(* Logix 5000 project; controller R5_CSS vendor 1 type 14 code 74 rev 19.11; software revision 19.01; part 13 of 20 *)
(* tags used below, declared in another part *)
   AC102A : ANALYTICAL;   // QUENCH WATER CONDUCTIVITY CONTROL
   bryans_Test4 : BOOL;
   CSS_Heartbeat : BOOL;
   CSS_OK_TO_RUN : BOOL;   // PRU_RUN_DISABLE 0 = Cannot Run 1 = OK to Run
   CSS_OK_TO_START : BOOL;   // PRU_START_DISABLE 0 = Cannot Start 1 = OK to Start
   LC303A : LEVEL_CONTROL;   // AQUEOUS PHASE OF PRIMARY SETTLER
   LC304 : LEVEL_CONTROL;   // SETTLER SECONDARY TANK INTERFACE LEVEL
   P101A : PUMP_CONTROL;
   P101B : PUMP_CONTROL;
   PC408 : PRESSURE_CONTROL;
   PRU_BLOWER_SEQ : INT;   // PRU BLOWER SEQUENCE NUMBER
   PRU_DELAY_REQ : INT;
   PRU_MaxTempDelayMin : REAL;
   PRU_MaxTempDelta : REAL;
   PRU_PT404 : REAL[10];
   PRU_PT404_Done : REAL[10];
   PRU_PT404_Max : REAL[10];
   PRU_RECIPE_LOAD : INT;
   PRU_RECIPE_LOAD_DLY : TIMER[10];
   PRU_RunDoneTemp : BOOL[32];
   PRU_RunDoneTime : BOOL[32];
   PRU_Running : BOOL[32];
   PRU_RunningMaxHrs : REAL;
   PRU_RunningMaxTempDelay : TIMER[10];
   PRU_RunningMinutePulse : TIMER[10];
   PRU_RunningTotalMin : COUNTER[10];
   PRU_START_REQ : INT;
   PRU_STARTDISABLE : DINT;   // PRU START DISABLE
   PRUA_CHANGE : INT;
   PRUA_CHANGE_OF_STATE : BOOL;
   PRUA_COMMS_TIMER : TIMER;
   PRUA_ECOOL : BOOL;
   PRUA_ECOOL_TON : TIMER;
   PRUA_HeartbeatCommsLoss : BOOL;
   PRUA_HeartbeatOffONS : BOOL;
   PRUA_HeartbeatOnONS : BOOL;
   PRUA_READ : INT[30];
   PRUA_START_REQ_ONS : BOOL[32];
   PRUA_WRITE : INT[40];
   PRUB_CHANGE : INT;
   PRUB_CHANGE_OF_STATE : BOOL;
   PRUB_COMMS_TIMER : TIMER;
   PRUB_ECOOL : BOOL;
   PRUB_ECOOL_TON : TIMER;
   PRUB_HeartbeatCommsLoss : BOOL;
   PRUB_HeartbeatOffONS : BOOL;
   PRUB_HeartbeatOnONS : BOOL;
   PRUB_READ : INT[30];
   PRUB_START_REQ_ONS : BOOL[32];
   PRUB_WRITE : INT[40];
   PRUC_CHANGE : INT;
   PRUC_CHANGE_OF_STATE : BOOL;
   PRUC_COMMS_TIMER : TIMER;
   PRUC_ECOOL : BOOL;
   PRUC_ECOOL_TON : TIMER;
   PRUC_HeartbeatCommsLoss : BOOL;
   PRUC_HeartbeatOffONS : BOOL;
   PRUC_HeartbeatOnONS : BOOL;
   PRUC_READ : INT[30];
   PRUC_START_REQ_ONS : BOOL[32];
   PRUC_WRITE : INT[40];
   TC101A : TEMP_CONTROL;   // QUENCH BASIN TRANSFER BASIN A TEMPERATURE CONTROL
   TC321A : TEMP_CONTROL;   // COALESCER OIL CHAMBER TRANSFER PUMP A TEMPERATURE TRANSMITTER
   TC321B : TEMP_CONTROL;   // COALESCER OIL CHAMBER TRANSFER PUMP B TEMPERATURE TRANSMITTER
   TMR_FAULT : DINT;
   UTL_Comms : DINT[3];
   UTL_CommsLossAlm : BOOL;
(* MainProgram, continued *)

ROUTINE PC408_FILL_IN_HERE   (* ladder *)
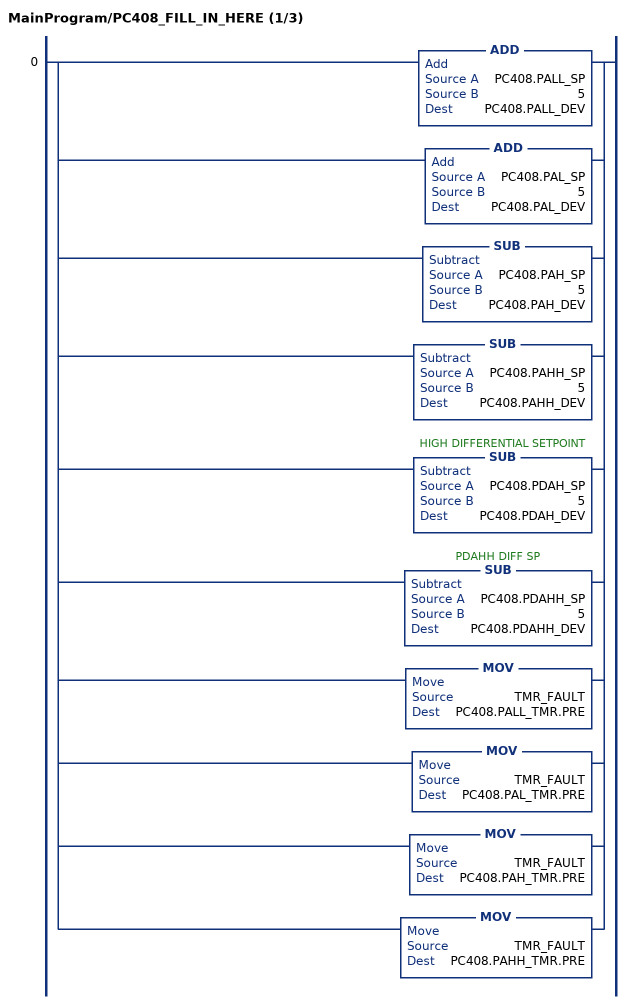
   0: [ADD(PC408.PALL_SP,5,PC408.PALL_DEV) ,ADD(PC408.PAL_SP,5,PC408.PAL_DEV) ,SUB(PC408.PAH_SP,5,PC408.PAH_DEV) ,SUB(PC408.PAHH_SP,5,PC408.PAHH_DEV) ,SUB(PC408.PDAH_SP,5,PC408.PDAH_DEV) ,SUB(PC408.PDAHH_SP,5,PC408.PDAHH_DEV) ,MOV(TMR_FAULT,PC408.PALL_TMR.PRE) ,MOV(TMR_FAULT,PC408.PAL_TMR.PRE) ,MOV(TMR_FAULT,PC408.PAH_TMR.PRE) ,MOV(TMR_FAULT,PC408.PAHH_TMR.PRE) ];
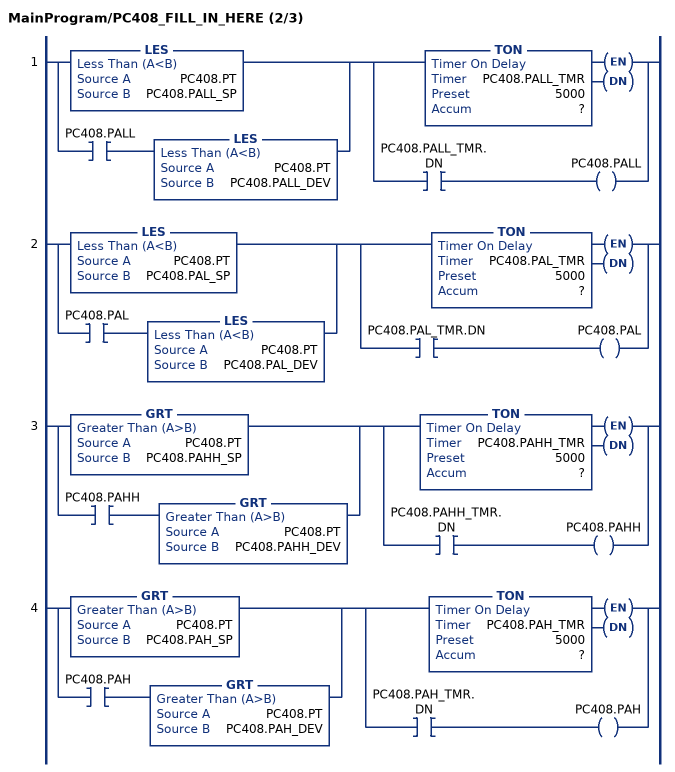
   1: [LES(PC408.PT,PC408.PALL_SP) ,XIC(PC408.PALL) LES(PC408.PT,PC408.PALL_DEV) ][TON(PC408.PALL_TMR,?,?) ,XIC(PC408.PALL_TMR.DN) OTE(PC408.PALL) ];
   2: [LES(PC408.PT,PC408.PAL_SP) ,XIC(PC408.PAL) LES(PC408.PT,PC408.PAL_DEV) ][TON(PC408.PAL_TMR,?,?) ,XIC(PC408.PAL_TMR.DN) OTE(PC408.PAL) ];
   3: [GRT(PC408.PT,PC408.PAHH_SP) ,XIC(PC408.PAHH) GRT(PC408.PT,PC408.PAHH_DEV) ][TON(PC408.PAHH_TMR,?,?) ,XIC(PC408.PAHH_TMR.DN) OTE(PC408.PAHH) ];
   4: [GRT(PC408.PT,PC408.PAH_SP) ,XIC(PC408.PAH) GRT(PC408.PT,PC408.PAH_DEV) ][TON(PC408.PAH_TMR,?,?) ,XIC(PC408.PAH_TMR.DN) OTE(PC408.PAH) ];
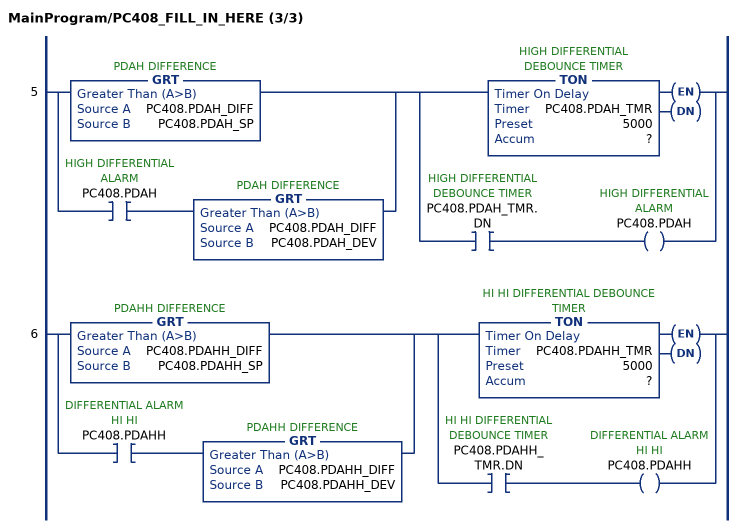
   5: [GRT(PC408.PDAH_DIFF,PC408.PDAH_SP) ,XIC(PC408.PDAH) GRT(PC408.PDAH_DIFF,PC408.PDAH_DEV) ][TON(PC408.PDAH_TMR,?,?) ,XIC(PC408.PDAH_TMR.DN) OTE(PC408.PDAH) ];
   6: [GRT(PC408.PDAHH_DIFF,PC408.PDAHH_SP) ,XIC(PC408.PDAHH) GRT(PC408.PDAHH_DIFF,PC408.PDAHH_DEV) ][TON(PC408.PDAHH_TMR,?,?) ,XIC(PC408.PDAHH_TMR.DN) OTE(PC408.PDAHH) ];
END_ROUTINE

ROUTINE PRU_STRTDIS   (* ladder *)
// PRU START DISABLE LOGIC
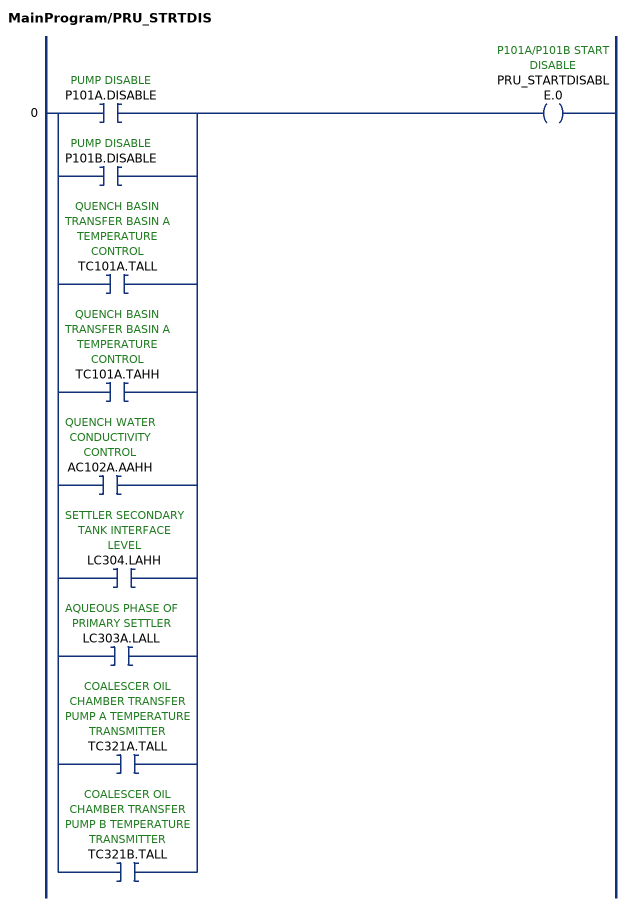
   0: [XIC(P101A.DISABLE) ,XIC(P101B.DISABLE) ,XIC(TC101A.TALL) ,XIC(TC101A.TAHH) ,XIC(AC102A.AAHH) ,XIC(LC304.LAHH) ,XIC(LC303A.LALL) ,XIC(TC321A.TALL) ,XIC(TC321B.TALL) ]OTE(PRU_STARTDISABLE.0);
END_ROUTINE

ROUTINE PRUA   (* ladder *)
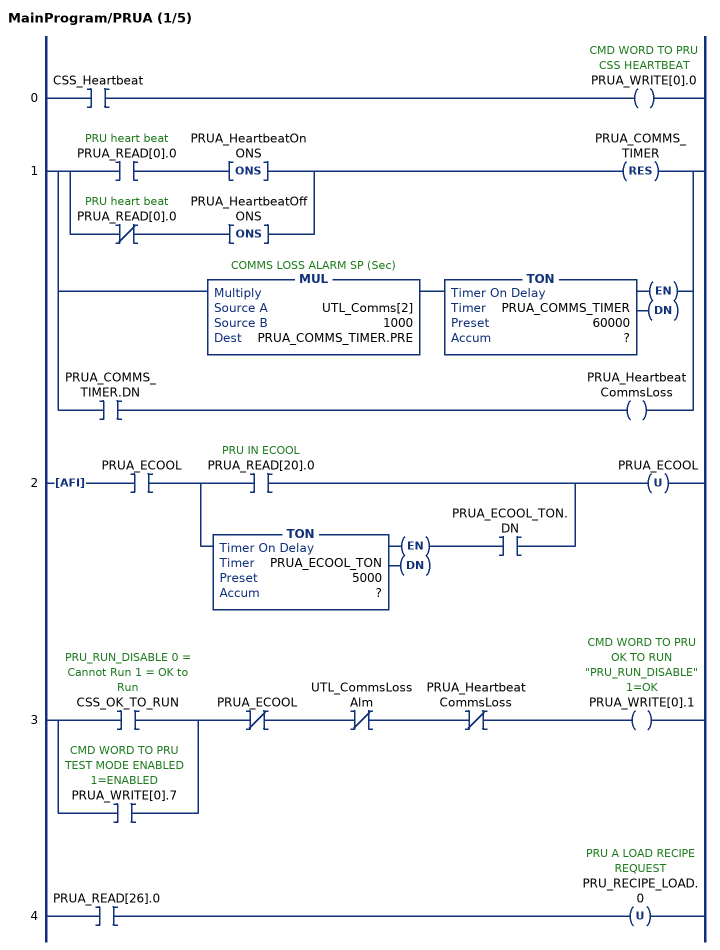
   0: XIC(CSS_Heartbeat)OTE(PRUA_WRITE[0].0);
   1: [[XIC(PRUA_READ[0].0) ONS(PRUA_HeartbeatOnONS) ,XIO(PRUA_READ[0].0) ONS(PRUA_HeartbeatOffONS) ] RES(PRUA_COMMS_TIMER) ,MUL(UTL_Comms[2],1000,PRUA_COMMS_TIMER.PRE) TON(PRUA_COMMS_TIMER,?,?) ,XIC(PRUA_COMMS_TIMER.DN) OTE(PRUA_HeartbeatCommsLoss) ];
   2: AFI()XIC(PRUA_ECOOL)[XIC(PRUA_READ[20].0) ,TON(PRUA_ECOOL_TON,?,?) XIC(PRUA_ECOOL_TON.DN) ]OTU(PRUA_ECOOL);
   3: [XIC(CSS_OK_TO_RUN) ,XIC(PRUA_WRITE[0].7) ]XIO(PRUA_ECOOL)XIO(UTL_CommsLossAlm)XIO(PRUA_HeartbeatCommsLoss)OTE(PRUA_WRITE[0].1);
   4: XIC(PRUA_READ[26].0)OTU(PRU_RECIPE_LOAD.0);
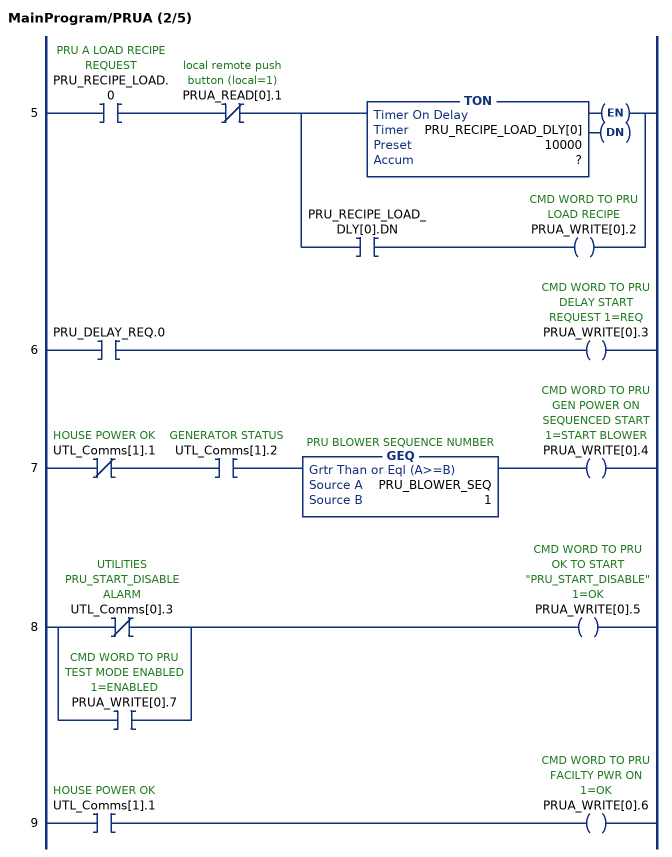
   5: XIC(PRU_RECIPE_LOAD.0)XIO(PRUA_READ[0].1)[TON(PRU_RECIPE_LOAD_DLY[0],?,?) ,XIC(PRU_RECIPE_LOAD_DLY[0].DN) OTE(PRUA_WRITE[0].2) ];
   6: XIC(PRU_DELAY_REQ.0)OTE(PRUA_WRITE[0].3);
   7: XIO(UTL_Comms[1].1)XIC(UTL_Comms[1].2)GEQ(PRU_BLOWER_SEQ,1)OTE(PRUA_WRITE[0].4);
   8: [XIO(UTL_Comms[0].3) ,XIC(PRUA_WRITE[0].7) ]OTE(PRUA_WRITE[0].5);
   9: XIC(UTL_Comms[1].1)OTE(PRUA_WRITE[0].6);
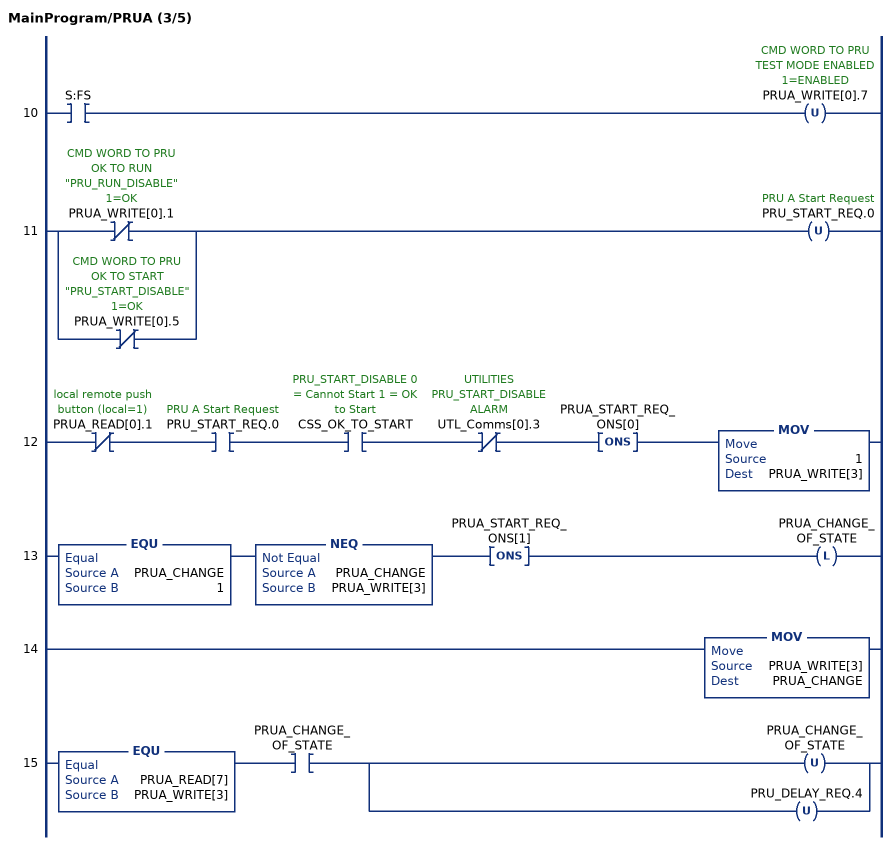
   10: XIC(S:FS)OTU(PRUA_WRITE[0].7);
   11: [XIO(PRUA_WRITE[0].1) ,XIO(PRUA_WRITE[0].5) ]OTU(PRU_START_REQ.0);
   12: XIO(PRUA_READ[0].1)XIC(PRU_START_REQ.0)XIC(CSS_OK_TO_START)XIO(UTL_Comms[0].3)ONS(PRUA_START_REQ_ONS[0])MOV(1,PRUA_WRITE[3]);
   13: EQU(PRUA_CHANGE,1)NEQ(PRUA_CHANGE,PRUA_WRITE[3])ONS(PRUA_START_REQ_ONS[1])OTL(PRUA_CHANGE_OF_STATE);
   14: MOV(PRUA_WRITE[3],PRUA_CHANGE);
   15: EQU(PRUA_READ[7],PRUA_WRITE[3])XIC(PRUA_CHANGE_OF_STATE)[OTU(PRUA_CHANGE_OF_STATE) ,OTU(PRU_DELAY_REQ.4) ];
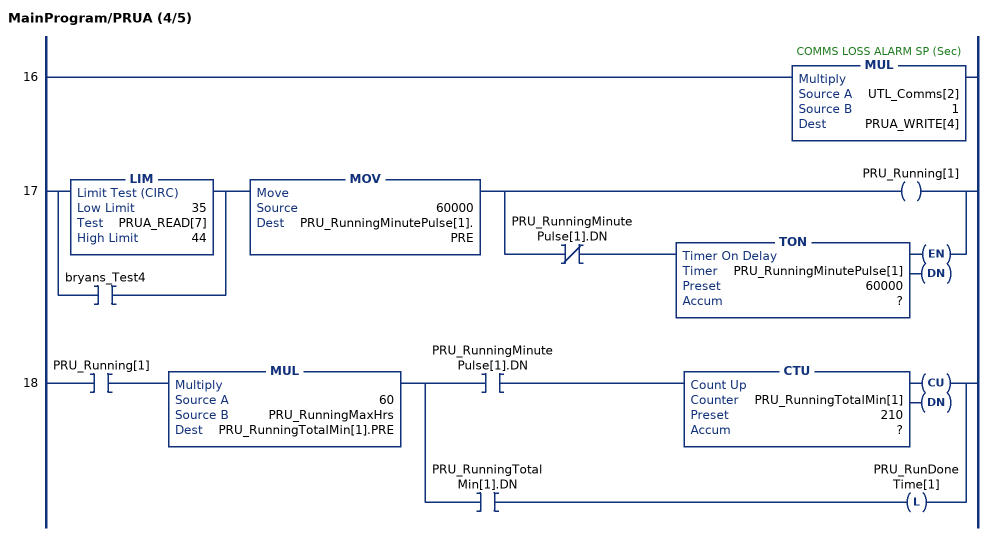
   16: MUL(UTL_Comms[2],1,PRUA_WRITE[4]);
   17: [LIM(35,PRUA_READ[7],44) ,XIC(bryans_Test4) ]MOV(60000,PRU_RunningMinutePulse[1].PRE)[OTE(PRU_Running[1]) ,XIO(PRU_RunningMinutePulse[1].DN) TON(PRU_RunningMinutePulse[1],?,?) ];
   18: XIC(PRU_Running[1])MUL(60,PRU_RunningMaxHrs,PRU_RunningTotalMin[1].PRE)[XIC(PRU_RunningMinutePulse[1].DN) CTU(PRU_RunningTotalMin[1],?,?) ,XIC(PRU_RunningTotalMin[1].DN) OTL(PRU_RunDoneTime[1]) ];
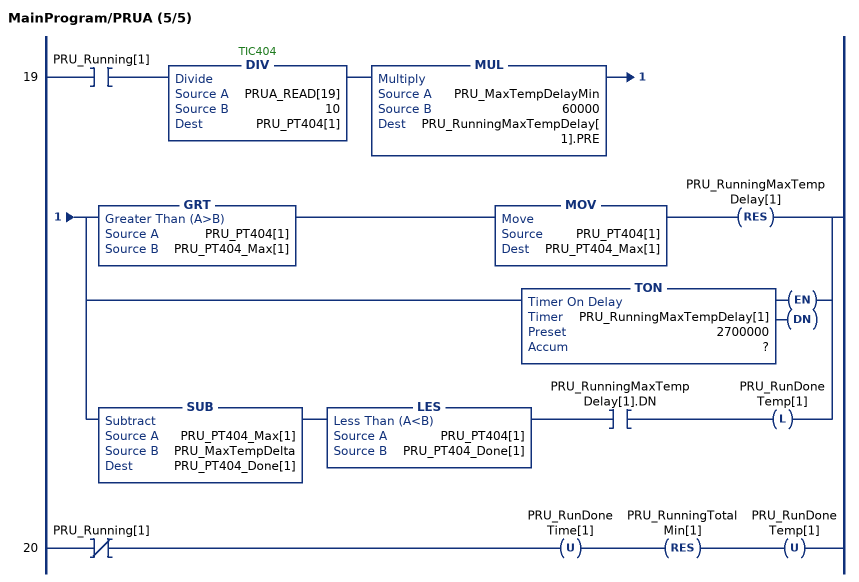
   19: XIC(PRU_Running[1])DIV(PRUA_READ[19],10,PRU_PT404[1])MUL(PRU_MaxTempDelayMin,60000,PRU_RunningMaxTempDelay[1].PRE)[GRT(PRU_PT404[1],PRU_PT404_Max[1]) MOV(PRU_PT404[1],PRU_PT404_Max[1]) RES(PRU_RunningMaxTempDelay[1]) ,TON(PRU_RunningMaxTempDelay[1],?,?) ,SUB(PRU_PT404_Max[1],PRU_MaxTempDelta,PRU_PT404_Done[1]) LES(PRU_PT404[1],PRU_PT404_Done[1]) XIC(PRU_RunningMaxTempDelay[1].DN) OTL(PRU_RunDoneTemp[1]) ];
   20: XIO(PRU_Running[1])OTU(PRU_RunDoneTime[1])RES(PRU_RunningTotalMin[1])OTU(PRU_RunDoneTemp[1]);
END_ROUTINE

ROUTINE PRUB   (* ladder *)
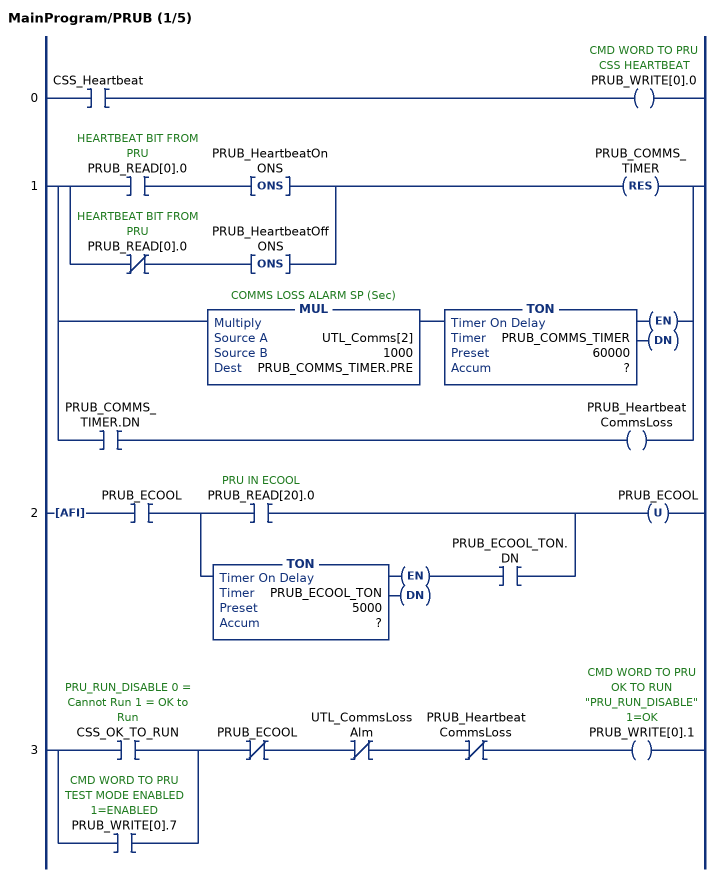
   0: XIC(CSS_Heartbeat)OTE(PRUB_WRITE[0].0);
   1: [[XIC(PRUB_READ[0].0) ONS(PRUB_HeartbeatOnONS) ,XIO(PRUB_READ[0].0) ONS(PRUB_HeartbeatOffONS) ] RES(PRUB_COMMS_TIMER) ,MUL(UTL_Comms[2],1000,PRUB_COMMS_TIMER.PRE) TON(PRUB_COMMS_TIMER,?,?) ,XIC(PRUB_COMMS_TIMER.DN) OTE(PRUB_HeartbeatCommsLoss) ];
   2: AFI()XIC(PRUB_ECOOL)[XIC(PRUB_READ[20].0) ,TON(PRUB_ECOOL_TON,?,?) XIC(PRUB_ECOOL_TON.DN) ]OTU(PRUB_ECOOL);
   3: [XIC(CSS_OK_TO_RUN) ,XIC(PRUB_WRITE[0].7) ]XIO(PRUB_ECOOL)XIO(UTL_CommsLossAlm)XIO(PRUB_HeartbeatCommsLoss)OTE(PRUB_WRITE[0].1);
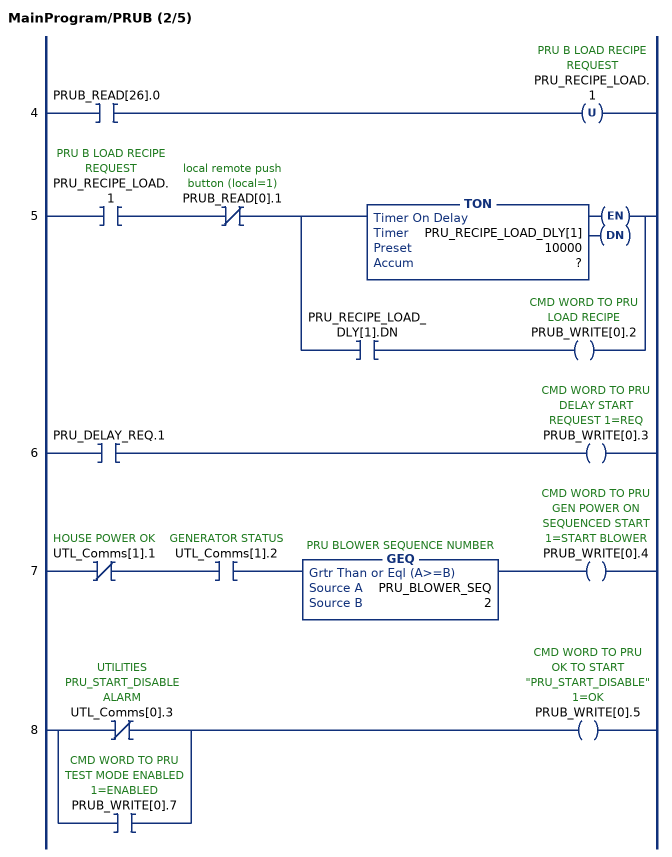
   4: XIC(PRUB_READ[26].0)OTU(PRU_RECIPE_LOAD.1);
   5: XIC(PRU_RECIPE_LOAD.1)XIO(PRUB_READ[0].1)[TON(PRU_RECIPE_LOAD_DLY[1],?,?) ,XIC(PRU_RECIPE_LOAD_DLY[1].DN) OTE(PRUB_WRITE[0].2) ];
   6: XIC(PRU_DELAY_REQ.1)OTE(PRUB_WRITE[0].3);
   7: XIO(UTL_Comms[1].1)XIC(UTL_Comms[1].2)GEQ(PRU_BLOWER_SEQ,2)OTE(PRUB_WRITE[0].4);
   8: [XIO(UTL_Comms[0].3) ,XIC(PRUB_WRITE[0].7) ]OTE(PRUB_WRITE[0].5);
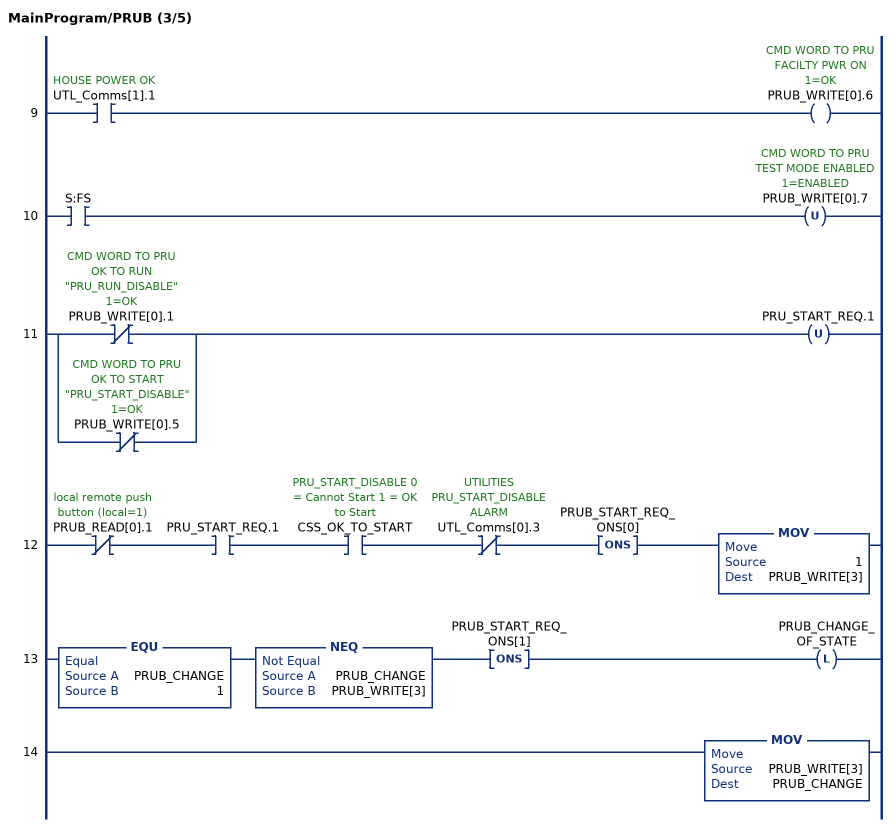
   9: XIC(UTL_Comms[1].1)OTE(PRUB_WRITE[0].6);
   10: XIC(S:FS)OTU(PRUB_WRITE[0].7);
   11: [XIO(PRUB_WRITE[0].1) ,XIO(PRUB_WRITE[0].5) ]OTU(PRU_START_REQ.1);
   12: XIO(PRUB_READ[0].1)XIC(PRU_START_REQ.1)XIC(CSS_OK_TO_START)XIO(UTL_Comms[0].3)ONS(PRUB_START_REQ_ONS[0])MOV(1,PRUB_WRITE[3]);
   13: EQU(PRUB_CHANGE,1)NEQ(PRUB_CHANGE,PRUB_WRITE[3])ONS(PRUB_START_REQ_ONS[1])OTL(PRUB_CHANGE_OF_STATE);
   14: MOV(PRUB_WRITE[3],PRUB_CHANGE);
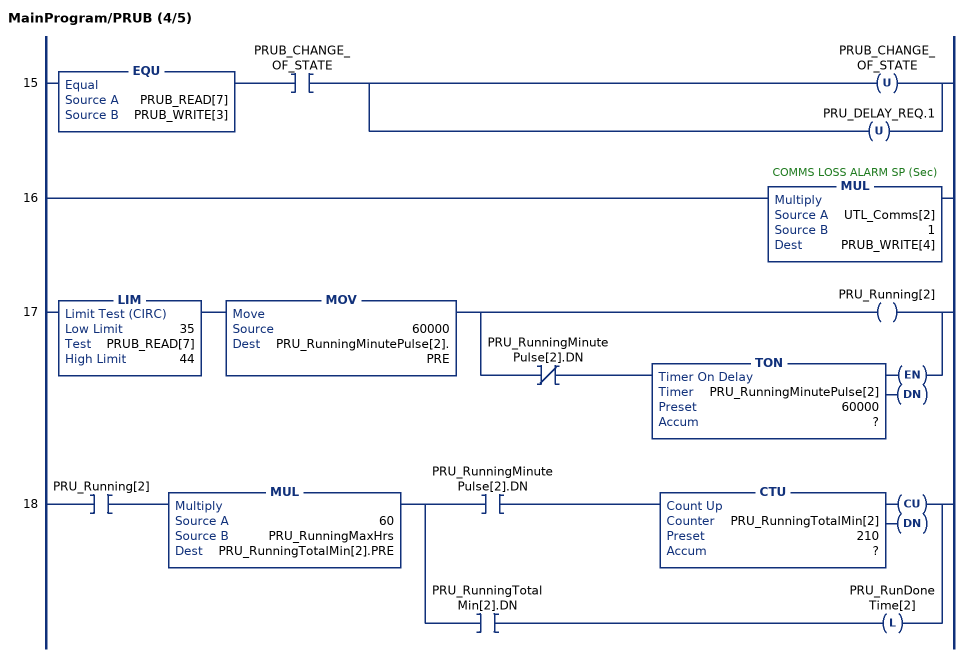
   15: EQU(PRUB_READ[7],PRUB_WRITE[3])XIC(PRUB_CHANGE_OF_STATE)[OTU(PRUB_CHANGE_OF_STATE) ,OTU(PRU_DELAY_REQ.1) ];
   16: MUL(UTL_Comms[2],1,PRUB_WRITE[4]);
   17: LIM(35,PRUB_READ[7],44)MOV(60000,PRU_RunningMinutePulse[2].PRE)[OTE(PRU_Running[2]) ,XIO(PRU_RunningMinutePulse[2].DN) TON(PRU_RunningMinutePulse[2],?,?) ];
   18: XIC(PRU_Running[2])MUL(60,PRU_RunningMaxHrs,PRU_RunningTotalMin[2].PRE)[XIC(PRU_RunningMinutePulse[2].DN) CTU(PRU_RunningTotalMin[2],?,?) ,XIC(PRU_RunningTotalMin[2].DN) OTL(PRU_RunDoneTime[2]) ];
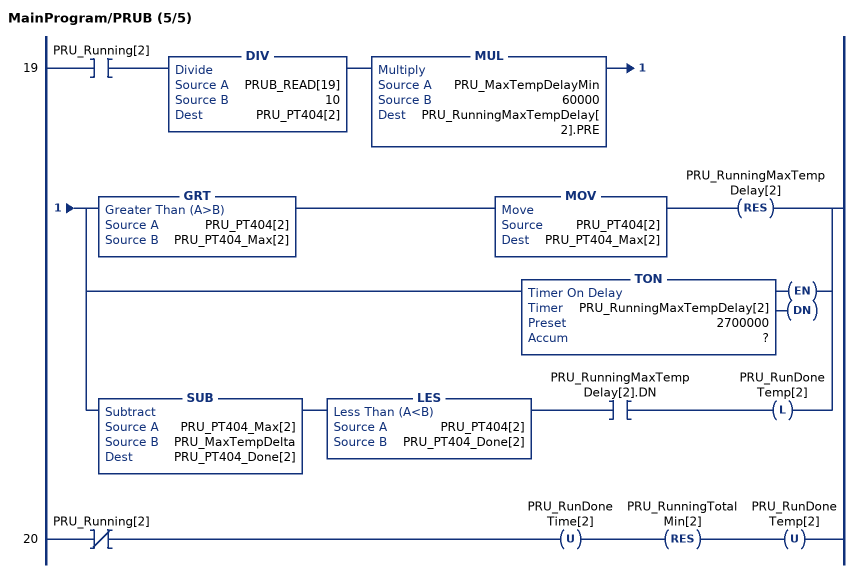
   19: XIC(PRU_Running[2])DIV(PRUB_READ[19],10,PRU_PT404[2])MUL(PRU_MaxTempDelayMin,60000,PRU_RunningMaxTempDelay[2].PRE)[GRT(PRU_PT404[2],PRU_PT404_Max[2]) MOV(PRU_PT404[2],PRU_PT404_Max[2]) RES(PRU_RunningMaxTempDelay[2]) ,TON(PRU_RunningMaxTempDelay[2],?,?) ,SUB(PRU_PT404_Max[2],PRU_MaxTempDelta,PRU_PT404_Done[2]) LES(PRU_PT404[2],PRU_PT404_Done[2]) XIC(PRU_RunningMaxTempDelay[2].DN) OTL(PRU_RunDoneTemp[2]) ];
   20: XIO(PRU_Running[2])OTU(PRU_RunDoneTime[2])RES(PRU_RunningTotalMin[2])OTU(PRU_RunDoneTemp[2]);
END_ROUTINE

ROUTINE PRUC   (* ladder *)
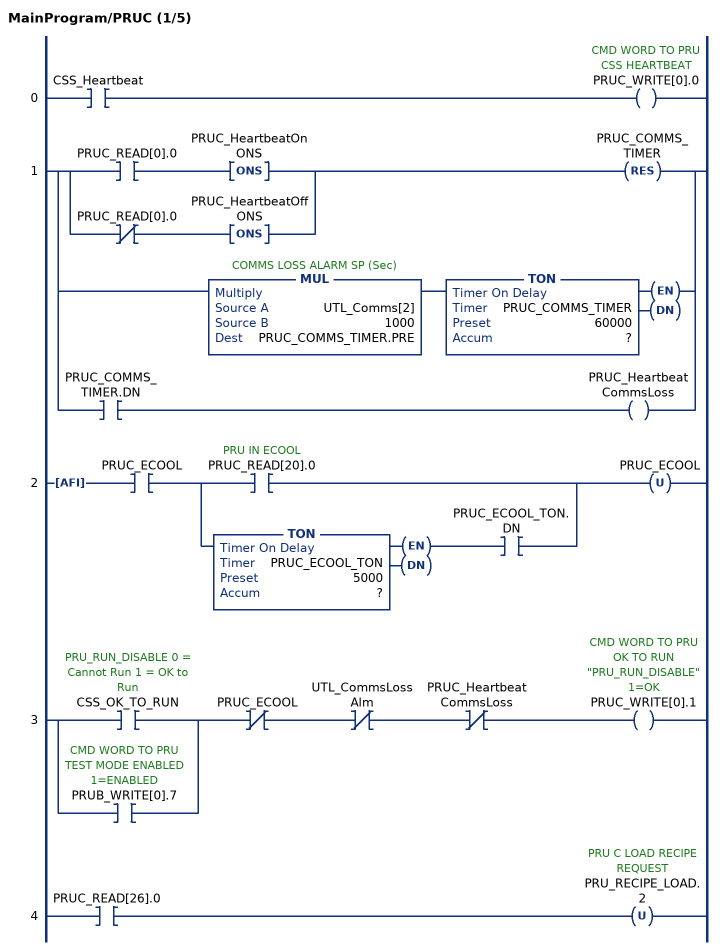
   0: XIC(CSS_Heartbeat)OTE(PRUC_WRITE[0].0);
   1: [[XIC(PRUC_READ[0].0) ONS(PRUC_HeartbeatOnONS) ,XIO(PRUC_READ[0].0) ONS(PRUC_HeartbeatOffONS) ] RES(PRUC_COMMS_TIMER) ,MUL(UTL_Comms[2],1000,PRUC_COMMS_TIMER.PRE) TON(PRUC_COMMS_TIMER,?,?) ,XIC(PRUC_COMMS_TIMER.DN) OTE(PRUC_HeartbeatCommsLoss) ];
   2: AFI()XIC(PRUC_ECOOL)[XIC(PRUC_READ[20].0) ,TON(PRUC_ECOOL_TON,?,?) XIC(PRUC_ECOOL_TON.DN) ]OTU(PRUC_ECOOL);
   3: [XIC(CSS_OK_TO_RUN) ,XIC(PRUB_WRITE[0].7) ]XIO(PRUC_ECOOL)XIO(UTL_CommsLossAlm)XIO(PRUC_HeartbeatCommsLoss)OTE(PRUC_WRITE[0].1);
   4: XIC(PRUC_READ[26].0)OTU(PRU_RECIPE_LOAD.2);
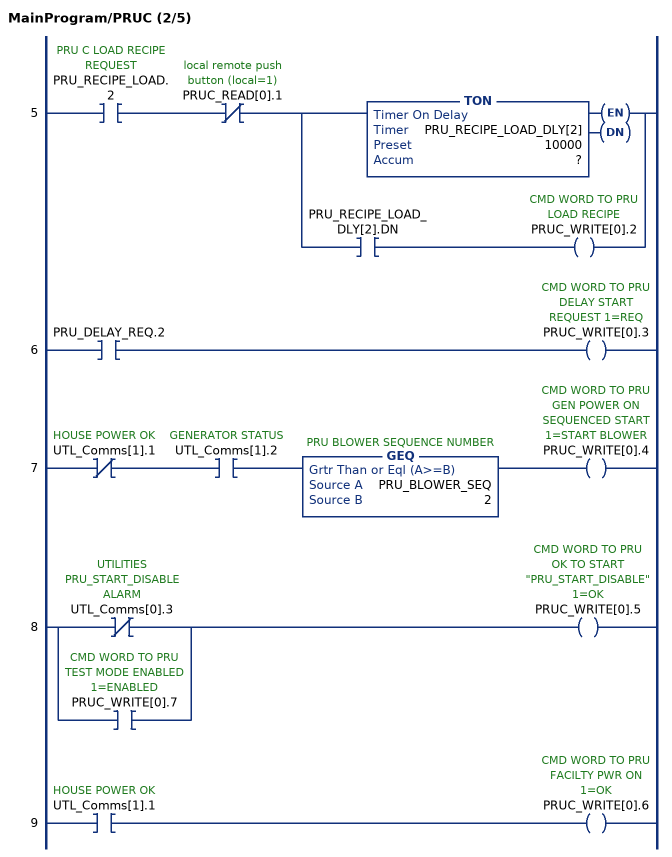
   5: XIC(PRU_RECIPE_LOAD.2)XIO(PRUC_READ[0].1)[TON(PRU_RECIPE_LOAD_DLY[2],?,?) ,XIC(PRU_RECIPE_LOAD_DLY[2].DN) OTE(PRUC_WRITE[0].2) ];
   6: XIC(PRU_DELAY_REQ.2)OTE(PRUC_WRITE[0].3);
   7: XIO(UTL_Comms[1].1)XIC(UTL_Comms[1].2)GEQ(PRU_BLOWER_SEQ,2)OTE(PRUC_WRITE[0].4);
   8: [XIO(UTL_Comms[0].3) ,XIC(PRUC_WRITE[0].7) ]OTE(PRUC_WRITE[0].5);
   9: XIC(UTL_Comms[1].1)OTE(PRUC_WRITE[0].6);
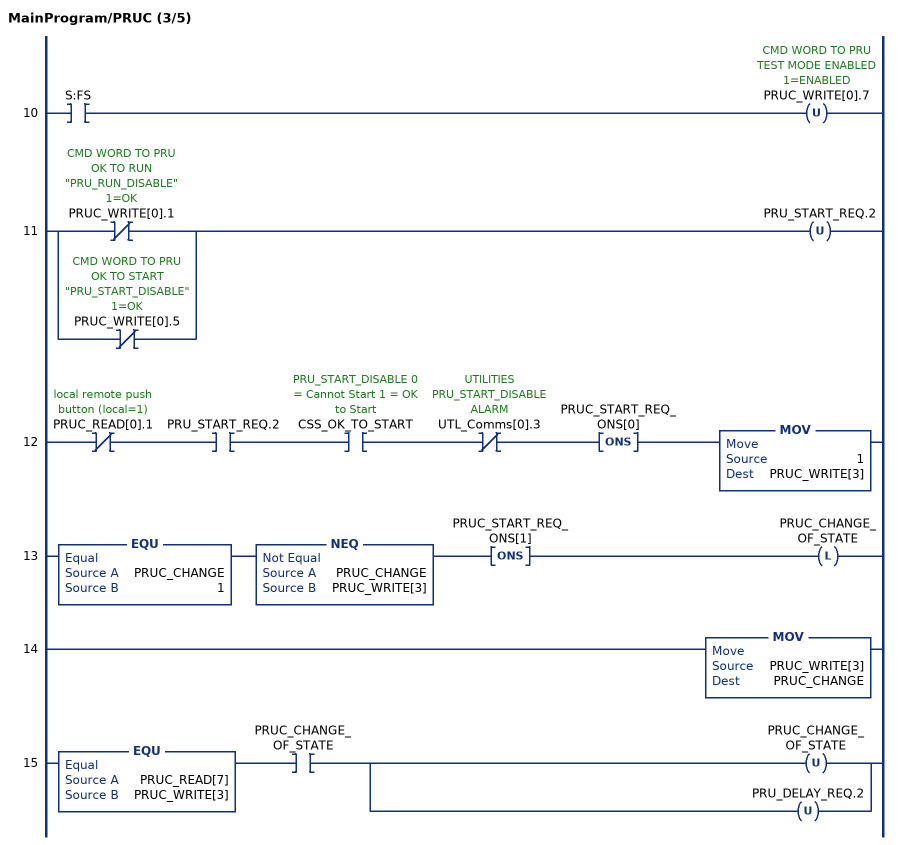
   10: XIC(S:FS)OTU(PRUC_WRITE[0].7);
   11: [XIO(PRUC_WRITE[0].1) ,XIO(PRUC_WRITE[0].5) ]OTU(PRU_START_REQ.2);
   12: XIO(PRUC_READ[0].1)XIC(PRU_START_REQ.2)XIC(CSS_OK_TO_START)XIO(UTL_Comms[0].3)ONS(PRUC_START_REQ_ONS[0])MOV(1,PRUC_WRITE[3]);
   13: EQU(PRUC_CHANGE,1)NEQ(PRUC_CHANGE,PRUC_WRITE[3])ONS(PRUC_START_REQ_ONS[1])OTL(PRUC_CHANGE_OF_STATE);
   14: MOV(PRUC_WRITE[3],PRUC_CHANGE);
   15: EQU(PRUC_READ[7],PRUC_WRITE[3])XIC(PRUC_CHANGE_OF_STATE)[OTU(PRUC_CHANGE_OF_STATE) ,OTU(PRU_DELAY_REQ.2) ];
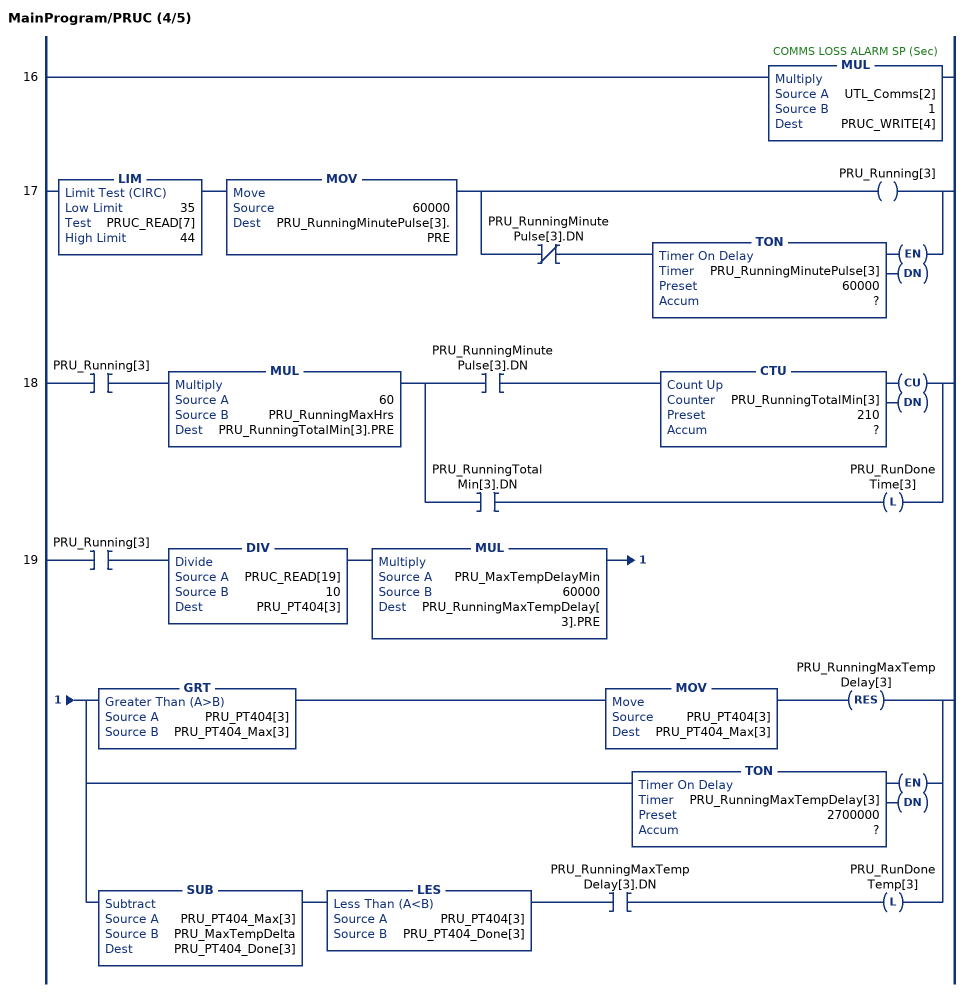
   16: MUL(UTL_Comms[2],1,PRUC_WRITE[4]);
   17: LIM(35,PRUC_READ[7],44)MOV(60000,PRU_RunningMinutePulse[3].PRE)[OTE(PRU_Running[3]) ,XIO(PRU_RunningMinutePulse[3].DN) TON(PRU_RunningMinutePulse[3],?,?) ];
   18: XIC(PRU_Running[3])MUL(60,PRU_RunningMaxHrs,PRU_RunningTotalMin[3].PRE)[XIC(PRU_RunningMinutePulse[3].DN) CTU(PRU_RunningTotalMin[3],?,?) ,XIC(PRU_RunningTotalMin[3].DN) OTL(PRU_RunDoneTime[3]) ];
   19: XIC(PRU_Running[3])DIV(PRUC_READ[19],10,PRU_PT404[3])MUL(PRU_MaxTempDelayMin,60000,PRU_RunningMaxTempDelay[3].PRE)[GRT(PRU_PT404[3],PRU_PT404_Max[3]) MOV(PRU_PT404[3],PRU_PT404_Max[3]) RES(PRU_RunningMaxTempDelay[3]) ,TON(PRU_RunningMaxTempDelay[3],?,?) ,SUB(PRU_PT404_Max[3],PRU_MaxTempDelta,PRU_PT404_Done[3]) LES(PRU_PT404[3],PRU_PT404_Done[3]) XIC(PRU_RunningMaxTempDelay[3].DN) OTL(PRU_RunDoneTemp[3]) ];
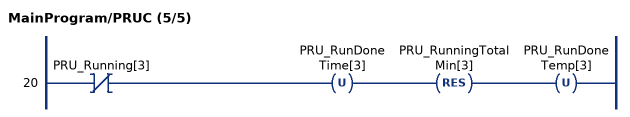
   20: XIO(PRU_Running[3])OTU(PRU_RunDoneTime[3])RES(PRU_RunningTotalMin[3])OTU(PRU_RunDoneTemp[3]);
END_ROUTINE
